Universal Robots PolyScope program: ad_pose_add_30.urp

Program ad_pose_add_30 (createdIn=3.2.19293 lastSavedIn=3.2.19293 directory=/programs installation=default robotSerialNumber=2015351391)
Calibrated DH parameters: a=[0.000352, -0.161198, -0.373486, 0.00005, 0.000049, 0]; d=[0.089268, 352.477598, -320.08558, -32.281492, 0.094939, 0.082518]; alpha=[1.570728, 0.001116, -0.003686, 1.571189, -1.570572, 0]; deltaTheta=[-0.000012, 1.181849, -1.491165, 0.309495, -0.000007, 0.000025]
Robot Program (runOnlyOnce=false motionType=MoveJ speed=1.047198 acceleration=1.396263 recalculateMotions=false)
  MoveJ speed 60 deg/s, acceleration 80 deg/s^2 (recalculateMotions=false)
    Waypoint refpoint: TCP in base x=37.665 y=237.35 z=361.758 mm, rx=1.555 ry=-2.5788 rz=-0.0637 rad; joints [101.136, -55.713, -105.274, -109.285, 97.536, 128.978] deg; flange x=54.196 y=241.2 z=485.607 mm, rx=1.555 ry=-2.5788 rz=-0.0639 rad
    Wait DigitalInput pin=Button; digitalValue=1
    Folder Calc_folder
      x := 250
      y := 120
      rz := 31
      offset := p[(x/1000),(y/1000),0,0,0,d2r(rz)]
      pick_pos := pose_add(refpoint,offset)
    MoveL speed 250 mm/s, acceleration 1200 mm/s^2 (recalculateMotions=false) feature=Base
      Waypoint 路点 (Variable): variable=pick_pos
